{attribute addProperty BoxType "AX5203-0000-0005-0005"}
{attribute addProperty Id "AT_xAT %I*ARRAY[0..2] OF AT_029F011596120MDTAT %Q*ARRAY[0..2] OF MDT_47A878CF96120WcStateAT %I*WcState_98A4DF7520.250InfoDataAT %I*InfoData_81099714160200"}
{attribute addProperty CRC "1275577876"}
{attribute addProperty SizeInBites "354"}
{attribute addProperty SizeInBytes "44.25"}
TYPE AX5203_D0280DF2 :
STRUCT
	{attribute addProperty Name "AT"}
	AT_x : ARRAY[0..2] OF AT_029F0115;
	{attribute addProperty Name "MDT"}
	MDT : ARRAY[0..2] OF MDT_47A878CF;
	{attribute addProperty Name "WcState"}
	WcState : WcState_98A4DF75;
	{attribute addProperty Name "InfoData"}
	InfoData : InfoData_81099714;
END_STRUCT
END_TYPE

(* stored: Version 1.2.0.0, ProductVersion 3.1.4024.9
   DUT AX5203_D0280DF2: Id {a265c9dd-38ae-4031-a42e-87777063dfb0} *)
